FUNCTION_BLOCK T_CartesianRobotManualMode EXTENDS T_NamedBase IMPLEMENTS I_PackMode
VAR
	_cartesianRobot : I_CartesianRobotModule;
END_VAR

METHOD Initialise
VAR_INPUT
	CartesianRobotModule : I_CartesianRobotModule; 
END_VAR
_cartesianRobot := CartesianRobotModule;
END_METHOD

END_FUNCTION_BLOCK

(* stored: Version 1.1.0.1, ProductVersion 3.1.4024.12
   POU T_CartesianRobotManualMode: Id {37544bab-a2c3-4917-9df6-e2192a9f0862}, SpecialFunc None
   Method Initialise: Id {036ea0e9-59f4-4026-9d9d-66a156616c38} *)
